// TwinCAT 3 PLC project PLC01
// ProgramVersion: 3.1.4026.12
// libraries:
//   Tc2_Standard, * (Beckhoff Automation GmbH)
//   Tc2_System, * (Beckhoff Automation GmbH)
// project tree:
//   DesignPatterns/ObserverPattern/classes/ AlarmLogger.TcPOU, VisitorHandler.TcPOU
//   DesignPatterns/ObserverPattern/gvls/ Gl1.TcGVL
//   DesignPatterns/ObserverPattern/Interfaces/ IVisitorHandler.TcIO, IVisitor.TcIO
//   DesignPatterns/ObserverPattern/programs/ ObserverPatternTest.TcPOU
//   DesignPatterns/StatePattern/classes/ FirstState.TcPOU, SecondState.TcPOU, StateManager.TcPOU
//   DesignPatterns/StatePattern/Interfaces/ Istate.TcIO
//   DesignPatterns/StatePattern/programs/ StatePatternTest.TcPOU
//   / MainTask.TcTTO
//   Tasks/ MAIN.TcPOU
// real-time tasks:
//   TASK MainTask: cycle T#20ms, priority 1, ADS port 351

CONFIGURATION PLC01
    RESOURCE PLC ON TwinCAT3
        TASK MainTask(INTERVAL := T#20ms, PRIORITY := 1);
        PROGRAM ObserverPatternTest WITH MainTask : ObserverPatternTest;
        PROGRAM StatePatternTest WITH MainTask : StatePatternTest;
    END_RESOURCE
END_CONFIGURATION

// ---- DesignPatterns/ObserverPattern/gvls/Gl1.TcGVL
{attribute 'qualified_only' := ''}
VAR_GLOBAL CONSTANT
	NUMOFSUBSCRIBERS: INT := 10;
END_VAR

// ---- DesignPatterns/ObserverPattern/Interfaces/IVisitorHandler.TcIO
INTERFACE IVisitorHandler

METHOD subscribe : BOOL
VAR_INPUT
	subscriber: IVisitor;
END_VAR
END_METHOD

METHOD unSubscribe : BOOL
VAR_INPUT
	subscriber: IVisitor;
END_VAR
END_METHOD

END_INTERFACE

// ---- DesignPatterns/ObserverPattern/Interfaces/IVisitor.TcIO
INTERFACE IVisitor

PROPERTY ActualValue : REAL
GET
END_GET
END_PROPERTY

METHOD updateValue : REAL
VAR_INPUT
	value: REAL;
END_VAR
END_METHOD

END_INTERFACE

// ---- DesignPatterns/StatePattern/Interfaces/Istate.TcIO
INTERFACE Istate

PROPERTY Description : STRING
GET
END_GET
END_PROPERTY

METHOD execute : BOOL
END_METHOD

END_INTERFACE

// ---- DesignPatterns/ObserverPattern/programs/ObserverPatternTest.TcPOU
PROGRAM ObserverPatternTest
VAR
	machine: VisitorHandler;
	AlarmLogger1: AlarmLogger;
	AlarmLogger2: AlarmLogger;
	AttachAlarmLogger1: BOOL;
	AttachAlarmLogger2: BOOL;
	DetachAlarmLogger1: BOOL;
	DetachAlarmLogger2: BOOL;
END_VAR

IF AttachAlarmLogger1 THEN
	AttachAlarmLogger1:= FALSE;
	machine.subscribe(AlarmLogger1);
END_IF


IF AttachAlarmLogger2 THEN
	AttachAlarmLogger2:= FALSE;
	machine.subscribe(AlarmLogger2);
END_IF


IF DetachAlarmLogger1 THEN
	DetachAlarmLogger1:= FALSE;
	machine.unSubscribe(AlarmLogger1);
END_IF

IF DetachAlarmLogger2 THEN
	DetachAlarmLogger2:= FALSE;
	machine.unSubscribe(AlarmLogger2);
END_IF



Machine.notify();
Machine.simulateValue();

END_PROGRAM

// ---- DesignPatterns/ObserverPattern/classes/VisitorHandler.TcPOU
FUNCTION_BLOCK VisitorHandler IMPLEMENTS IVisitorHandler
VAR
	_subscribers: ARRAY[1..Gl1.NUMOFSUBSCRIBERS] OF IVisitor;
	_ActualTemperature: REAL;
END_VAR

METHOD PRIVATE checkSubscriber : BOOL
VAR_INPUT
	subscriber: IVisitor;
END_VAR
VAR
	index: INT;
END_VAR
RETURN (subscriber =0);

checkSubscriber:= TRUE;
FOR index:=1 TO Gl1.NUMOFSUBSCRIBERS BY 1 DO
	IF THIS^._subscribers[index]=subscriber 	THEN
		RETURN;
	END_IF
END_FOR 
checkSubscriber:= FALSE;
END_METHOD

METHOD notify : BOOL
VAR
	index: INT;
END_VAR
FOR index :=1 TO Gl1.NUMOFSUBSCRIBERS BY 1 DO 
	IF THIS^._subscribers[index]<>0 THEN
		THIS^._subscribers[index].updateValue(THIS^._ActualTemperature);
	END_IF	
END_FOR
END_METHOD

METHOD simulateValue
THIS^._ActualTemperature:= (THIS^._ActualTemperature +0.001) ;
END_METHOD

METHOD subscribe : BOOL
VAR_INPUT
	subscriber: IVisitor;
END_VAR
VAR
	index: INT;
END_VAR

RETURN (subscriber =0 OR checkSubscriber(subscriber));

FOR index :=1 TO Gl1.NUMOFSUBSCRIBERS BY 1 DO 
	IF THIS^._subscribers[index]=0 THEN
		THIS^._subscribers[index]:=subscriber;
		subscribe:= TRUE;
		RETURN;
	END_IF
END_FOR
END_METHOD

METHOD unSubscribe : BOOL
VAR_INPUT
	subscriber: IVisitor;
END_VAR
VAR
	index: INT;
END_VAR
RETURN (subscriber =0);

FOR index :=1 TO Gl1.NUMOFSUBSCRIBERS BY 1 DO 
	IF THIS^._subscribers[index]= subscriber THEN
		THIS^._subscribers[index]:=0;
		unSubscribe:=TRUE;
		RETURN;
	END_IF
END_FOR
END_METHOD

END_FUNCTION_BLOCK

// ---- DesignPatterns/ObserverPattern/classes/AlarmLogger.TcPOU
FUNCTION_BLOCK AlarmLogger IMPLEMENTS IVisitor
VAR
	_value: REAL;
END_VAR

PROPERTY actualValue : REAL
GET
ActualValue:=this^._value;
END_GET
END_PROPERTY

METHOD updateValue : REAL
VAR_INPUT
	value: REAL;
END_VAR
this^._value:= value;
END_METHOD

END_FUNCTION_BLOCK

// ---- DesignPatterns/StatePattern/programs/StatePatternTest.TcPOU
PROGRAM StatePatternTest
VAR
	stateManger: StateManager;
	firststate: FirstState;
	secondState: SecondState;
	stateslist: ARRAY[1..2] OF Istate:=[firststate,secondState];
END_VAR


stateManger(statelist := stateslist);
stateManger.RunProcess();

END_PROGRAM

// ---- DesignPatterns/StatePattern/classes/StateManager.TcPOU
FUNCTION_BLOCK StateManager
VAR_IN_OUT
	statelist: ARRAY[*] OF IState;
END_VAR
VAR
	index: INT:=1;
	message: String;
END_VAR

METHOD RunProcess : BOOL
IF THIS^.statelist[index]<>0 THEN
	IF THIS^.statelist[index].execute() THEN
		IF index<= SIZEOF(statelist)-1 THEN		
			index:=index+1;
		ELSE
			index:=1;
		END_IF
	END_IF
	message:= THIS^.statelist[index].Description;
END_IF
END_METHOD

END_FUNCTION_BLOCK

// ---- DesignPatterns/StatePattern/classes/FirstState.TcPOU
FUNCTION_BLOCK FirstState IMPLEMENTS Istate
VAR
	stateFinished: BOOL;
	_description: STRING := 'FirstState';
END_VAR

PROPERTY Description : STRING
GET
Description:= _description;
END_GET
END_PROPERTY

METHOD execute : BOOL
IF NOT stateFinished THEN 
	THIS^();
END_IF

execute:= stateFinished;
END_METHOD

///FB_Init is always available implicitly and it is used primarily for initialization.
///The return value is not evaluated. For a specific influence, you can also declare the
///methods explicitly and provide additional code there with the standard initialization
///code. You can evaluate the return value.
METHOD FB_Init : BOOL
VAR_INPUT
	/// TRUE: the retain variables are initialized (reset warm / reset cold)
	bInitRetains: BOOL;
	/// TRUE: the instance will be copied to the copy code afterward (online change) 
	bInCopyCode: BOOL;
END_VAR
END_METHOD

END_FUNCTION_BLOCK

// ---- DesignPatterns/StatePattern/classes/SecondState.TcPOU
FUNCTION_BLOCK SecondState IMPLEMENTS Istate
VAR
	stateFinished: BOOL;
	_description: STRING := 'SecondState';
END_VAR

PROPERTY Description : STRING
GET
Description:= _description;
END_GET
END_PROPERTY

METHOD execute : BOOL
IF NOT stateFinished THEN 
	THIS^();
END_IF

execute:= stateFinished;
END_METHOD

///FB_Init is always available implicitly and it is used primarily for initialization.
///The return value is not evaluated. For a specific influence, you can also declare the
///methods explicitly and provide additional code there with the standard initialization
///code. You can evaluate the return value.
METHOD FB_Init : BOOL
VAR_INPUT
	/// TRUE: the retain variables are initialized (reset warm / reset cold)
	bInitRetains: BOOL;
	/// TRUE: the instance will be copied to the copy code afterward (online change) 
	bInCopyCode: BOOL;
END_VAR
END_METHOD

END_FUNCTION_BLOCK

// ---- Tasks/MAIN.TcPOU
PROGRAM MAIN
VAR
END_VAR

END_PROGRAM
